{attribute addProperty BoxType "AT2050-0500-0023"}
{attribute addProperty Id "A_0090_AT2050_5501_0019_AT2050_5501AT2050_C5E5984862678.25"}
{attribute addProperty CRC "2647976699"}
{attribute addProperty SizeInBites "626"}
{attribute addProperty SizeInBytes "78.25"}
TYPE A_0054_AT2050_0500_0023_9DD4EAFB EXTENDS AT2050_BA5A9548 :
STRUCT
	{attribute addProperty Name "A_0090_AT2050_5501_0019_AT2050_5501"}
	A_0090_AT2050_5501_0019_AT2050_5501 : AT2050_C5E59848;
END_STRUCT
END_TYPE

(* stored: Version 1.2.0.0, ProductVersion 3.1.4024.9
   DUT A_0054_AT2050_0500_0023_9DD4EAFB: Id {bfcad69f-a2b0-4020-ab48-ead0d9008e83} *)
